// TIA Portal V20 export
DATA_BLOCK "LPFE_MainBuffer"   // DB243
TITLE = Buffer of RequestOrderInfo messages
// Buffer to store digital/value messages (5,6) until distributed
// stored: Access Published, MemoryReserve 100, Namespace PFE
   VAR
      buffer { ExternalAccessible := 'False'; ExternalVisible := 'False'; ExternalWritable := 'False'} : Array[0.._.LE_NUMBER_MESSAGES_MAIN_BUFFER] of "LPFE_typePFEDataReqEnvelope";   // Buffer where digital/alarm messages are taken from
      mgmtBuffer { ExternalAccessible := 'False'; ExternalVisible := 'False'; ExternalWritable := 'False'} : "LPFE_typeMsgBuffer";   // Mgmt Structure of buffer where digital/alarm messages are taken from
      mainBufferBlocked { ExternalAccessible := 'False'; ExternalVisible := 'False'; ExternalWritable := 'False'} : Bool;   // Main Buffer blocked due to a Reset Event
      resetReceived { ExternalAccessible := 'False'; ExternalVisible := 'False'; ExternalWritable := 'False'} : Bool;   // TRUE: Reset command received
      sendResourceEventsAfterReset { ExternalAccessible := 'False'; ExternalVisible := 'False'; ExternalWritable := 'False'} : Bool;   // TRUE: boolean used to trigger the sending of resource events after a reset sequence
      resourceSent { ExternalAccessible := 'False'; ExternalVisible := 'False'; ExternalWritable := 'False'} : Bool;   // TRUE: flag to indicate that all the resource events where sent after a reset sequence
   END_VAR
BEGIN
END_DATA_BLOCK
